TYPE Vec4b : ARRAY[1..4] OF BOOl; END_TYPE

(* stored: Version 1.1.0.1, ProductVersion 3.1.4024.12
   DUT Vec4b: Id {da60e75d-21a5-4d9e-a85a-54bf25c4bcfe} *)
